(* LS Electric XG5000 project: HomingWalkThrough *)
(* PLC LSPLC *)
(* module base 0 slot 0: Input/Output Module:XEM-DN/DP32HP (DC 24V Input, Transistor Output, 32 Contacts) *)
(* module base 0 slot 1: Internal Positioning:XBF-PO06E (Open Collector Type, 6 Axis) *)
VAR_GLOBAL
    A1_Home_Done : BOOL;
    A1_ORG_Done : BOOL;
    A1_ORG_Stat : UINT;
    Axis1_RST : XPM_RST;
    Dog_SW AT %IX0.0.5 : BOOL;
    High_LIMIT AT %IX0.0.6 : BOOL;
    Home_SW AT %IX0.0.4 : BOOL;
    Low_LIMIT AT %IX0.0.3 : BOOL;
    ResetAxis AT %IX0.0.1 : BOOL; (* Send Axis reset command to motion CPU *)
    SeekHome AT %IX0.0.0 : BOOL; (* initiate homing routine *)
    Stop AT %IX0.0.2 : BOOL; (* Immediate Stop (No decel time) *)
END_VAR

PROGRAM HomeTheAxis (* task: Scan Program *)
VAR
    A1_FLT_Done : BOOL;
    A1_FLT_Stat : UINT;
    Axis1 : XPM_ORG;
    Axis1_EMG : XPM_EMG;
    Axis1_FLT_Home : APM_FLT;
    Axis1_FLT_Home1 : XPM_FLT;
    Axis1_ORG : XPM_ORG;
    Axis1_PRS : XPM_PRS;
    Axis1_STP : XPM_STP;
    Change_Origin : BOOL;
    Create_New_Position : BOOL;
    Create_Origin : BOOL;
    New_ORG_value : DINT;
    New_Position_value : DINT;
    XAxis_EMG1 : XPM_EMG;
END_VAR
VAR_EXTERNAL
    A1_Home_Done : BOOL;
    A1_ORG_Done : BOOL;
    A1_ORG_Stat : UINT;
    Axis1_RST : XPM_RST;
    ResetAxis : BOOL; (* AT %IX0.0.1 *) (* Send Axis reset command to motion CPU *)
    SeekHome : BOOL; (* AT %IX0.0.0 *) (* initiate homing routine *)
    Stop : BOOL; (* AT %IX0.0.2 *) (* Immediate Stop (No decel time) *)
END_VAR

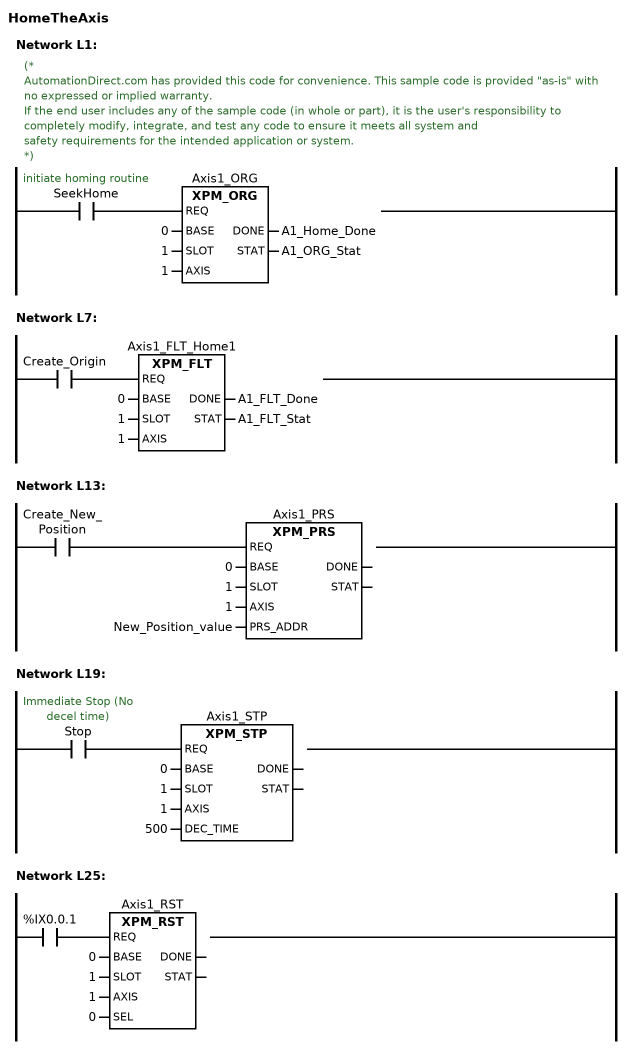
(* ( * / AutomationDirect.com has provided this code for convenience. This sample code is provided "as-is" with no expressed or implied warranty. / If the end user includes any of the sample code (in whole or part), it is the user's responsibility to completely modify, integrate, and test any code to ensure it meets all system and / safety requirements for the intended application or system. / * ) *)
(* Rung L1 *)
Axis1_ORG(REQ := SeekHome, BASE := 0, SLOT := 1, AXIS := 1, DONE => A1_Home_Done, STAT => A1_ORG_Stat);
(* Rung L7 *)
Axis1_FLT_Home1(REQ := Create_Origin, BASE := 0, SLOT := 1, AXIS := 1, DONE => A1_FLT_Done, STAT => A1_FLT_Stat);
(* Rung L13 *)
Axis1_PRS(REQ := Create_New_Position, BASE := 0, SLOT := 1, AXIS := 1, PRS_ADDR := New_Position_value);
(* Rung L19 *)
Axis1_STP(REQ := Stop, BASE := 0, SLOT := 1, AXIS := 1, DEC_TIME := 500);
(* Rung L25 *)
Axis1_RST(REQ := %IX0.0.1, BASE := 0, SLOT := 1, AXIS := 1, SEL := 0);
END_PROGRAM